PROGRAM PRG_Cryo
VAR
    fb_Cryo_ROT : FB_MotionStage;
    fb_Cryo_X : FB_MotionStage;
    fb_Cryo_Y : FB_MotionStage;
    fb_Cryo_Z : FB_MotionStage;
    bInit : BOOl := TRUE;
END_VAR

IF ( bInit) THEN
    bInit := FALSE;
    Main.M46.bHardwareEnable := TRUE;
    Main.M46.bPowerSelf := TRUE;
    Main.M46.nBrakeMode := ENUM_StageBrakeMode.NO_BRAKE;
    Main.M46.nEnableMode := ENUM_StageEnableMode.DURING_MOTION;

    Main.M47.bHardwareEnable := TRUE;
    Main.M47.bPowerSelf := TRUE;
    Main.M47.nBrakeMode := ENUM_StageBrakeMode.NO_BRAKE;
    Main.M47.nEnableMode := ENUM_StageEnableMode.DURING_MOTION;

    Main.M48.bHardwareEnable := TRUE;
    Main.M48.bPowerSelf := TRUE;
    Main.M48.nBrakeMode := ENUM_StageBrakeMode.NO_BRAKE;
    Main.M48.nEnableMode := ENUM_StageEnableMode.DURING_MOTION;

    Main.M49.bHardwareEnable := TRUE;
    Main.M49.bPowerSelf := TRUE;
    Main.M49.nBrakeMode := ENUM_StageBrakeMode.NO_BRAKE;
    Main.M49.nEnableMode := ENUM_StageEnableMode.DURING_MOTION;
END_IF


//EPS??

fb_Cryo_X(stMotionStage:=Main.M46);
fb_Cryo_Y(stMotionStage:=Main.M47);
fb_Cryo_Z(stMotionStage:=Main.M48);
fb_Cryo_ROT(stMotionStage:=Main.M49);

END_PROGRAM

(* stored: Version 1.1.0.1, ProductVersion 3.1.4022.18
   POU PRG_Cryo: Id {d8649ca7-c26e-4e28-a279-17f291a3cb8e}, SpecialFunc None *)
